// TwinCAT 3 PLC project AnalogMotorControl
// ProgramVersion: 3.1.4024.0
// libraries:
//   Tc2_Math, * (Beckhoff Automation GmbH)
//   Tc2_Standard, * (Beckhoff Automation GmbH)
//   Tc2_System, * (Beckhoff Automation GmbH)
//   Tc2_Utilities, * (Beckhoff Automation GmbH)
//   Tc3_Module, * (Beckhoff Automation GmbH)
// project tree:
//   / PlcTask.TcTTO
//   POUs/ AnalogMotorDriver.TcPOU, MAIN.TcPOU
// real-time tasks:
//   TASK PlcTask: cycle T#100us, priority 20, ADS port 350
// I/O:
//   DEVICE Device 2 (EtherCAT), AmsNetId 141.212.76.55.3.1
//     Term 1 (EK1100) [EK1100 EtherCAT Coupler (2A E-Bus)]
//       Term 2 (EL4038) [EL4038 8Ch. Ana. Output +/-10V, 12bit]
//       Term 3 (EL3174) [EL3174 4Ch. Ana. Input +/-10V Diff., +/-20mA SingleEnded, 16 Bit]
//       Term 4 (EL5122) [EL5122 2Ch. Inc. Encoder 5V (2xAB TTL)]
//       Term 5 (EL9011) [EL9011 End Terminal]
// variable links:
//   AnalogMotorControl/AnalogMotorControl Instance <-> Device 2 (EtherCAT)/Term 1 (EK1100)/Term 2 (EL4038)
//     PlcTask Outputs/MAIN.AM_Driver.nNegAnalogOutput <-> AO Outputs Channel 2/Analog output
//     PlcTask Outputs/MAIN.AM_Driver.nPosAnalogOutput <-> AO Outputs Channel 1/Analog output
//     PlcTask Outputs/MAIN.AM_Driver.nZeroRefAnalogOutput <-> AO Outputs Channel 3/Analog output

CONFIGURATION AnalogMotorControl
    RESOURCE PLC ON TwinCAT3
        TASK PlcTask(INTERVAL := T#100us, PRIORITY := 20);
        PROGRAM MAIN WITH PlcTask : MAIN;
    END_RESOURCE
END_CONFIGURATION

// ---- POUs/MAIN.TcPOU
PROGRAM MAIN
VAR
	AM_Driver : AnalogMotorDriver; 
	fbSystemTime : GETSYSTEMTIME; 
	lowerHalf : UDINT; // Lower 32 bits 
	upperHalf : UDINT; // Upper 32 bits 
	fullTime : ULINT; // Combined 64 bits
	currentTimeSeconds : LREAL; 
	elapsedSeconds : LREAL; 
	
	bInitialTimeSet : BOOL := FALSE; 
	initialTimeSeconds : LREAL; // To store initial time for reference 
	
	// Output values for sine 
	rSineSignal : LREAL; 
	nPosOutputCommand : INT; 
	nNegOutputCommand : INT; 
	
END_VAR

// Poll the current system time 
fbSystemTime();
lowerHalf := fbSystemTime.timeLoDW; 
upperHalf := fbSystemTime.timeHiDW; 

fullTime := SHL(UDINT_TO_ULINT(upperHalf), 32) OR UDINT_TO_ULINT(lowerHalf); 
currentTimeSeconds := ULINT_TO_LREAL(fullTime) / 10000000.0; 

// Check to see if we need to set our initial condition. 
IF NOT bInitialTimeSet THEN
	initialTimeSeconds := currentTimeSeconds; 
	bInitialTimeSet := TRUE; 
END_IF

// Then get the DT 
elapsedSeconds := currentTimeSeconds - initialTimeSeconds; 

// Finally, pass the sine value to see what's up 
rSineSignal := 2 * SIN(elapsedSeconds * 2 * 3.14); 
AM_Driver(rCommandVoltage := rSineSignal); 
nPosOutputCommand := AM_Driver.nPosAnalogOutput; 
nNegOutputCommand := AM_Driver.nNegAnalogOutput;

END_PROGRAM

// ---- POUs/AnalogMotorDriver.TcPOU
FUNCTION_BLOCK AnalogMotorDriver
VAR_INPUT
	// Nominally, respect requested command voltage between (-10)-10V, i.e. if rCommandVoltage
	// is 5, then the output on the channel should be 5V. However, we can alternatively 
	// Request voltage in normalized mode, which considers rCommandVoltage as a 
	// normalized signal between (-1)-1. To enable this mode, set the bUseNormalizedScale
	// flag, which is defaulted to false. When normalized signals are used, the user can additionally 
	// specify whether normalized commands map to (-10)-10V, or (-5)-5V; the latter is triggered
	// when bUseHalfScale is set to TRUE. 
	rCommandVoltage : REAL;
	bUseNormalizedScale : BOOL := FALSE;
	bUseHalfScale : BOOL := FALSE; 
END_VAR
VAR_OUTPUT
	nPosAnalogOutput AT %Q* : INT; 
	nNegAnalogOutput AT %Q* : INT; 
	nZeroRefAnalogOutput AT %Q* : INT; 
	bOutputInError : BOOL; 
END_VAR
VAR
	nTEN_VOLT_AMPLITUDE : INT := 32767; 
	nFIVE_VOLT_AMPLITUDE : INT := 16383;
END_VAR

IF NOT bUseNormalizedScale THEN 
	
	// In this case we were passed a raw voltage signal. 
	// Should check to see if scaling is appropriate, etc. 
	IF ABS(rCommandVoltage) > 10 THEN
		bOutputInError := TRUE; 
		RETURN; 
	END_IF
	
	nPosAnalogOutput := REAL_TO_INT(rCommandVoltage * nTEN_VOLT_AMPLITUDE / 10.0);
	nNegAnalogOutput := -1 * nPosAnalogOutput;  
	
	bOutputInError := FALSE;

ELSE 
	
	// Again check if argument is valid
	IF ABS(rCommandVoltage) > 1 THEN 
		bOutputInError := TRUE; 
		RETURN;
	END_IF
	
	// Check to see if we should use the half scale. 
	IF bUseHalfScale THEN
		nPosAnalogOutput := REAL_TO_INT(rCommandVoltage * nFIVE_VOLT_AMPLITUDE); 
	ELSE
		nPosAnalogOutput := REAL_TO_INT(rCommandVoltage * nTEN_VOLT_AMPLITUDE); 
	END_IF
	
	nNegAnalogOutput := -1 * nPosAnalogOutput;  
	bOutputInError := FALSE; 
	
END_IF

END_FUNCTION_BLOCK
